PROGRAM MOTORS
VAR
	
END_VAR

Axis_MAIN(sName:='MAIN');
Axis_SUPPLY(sNAme:='SUPPLY');
Axis_JACK1(sNAme:='JACK1');

END_PROGRAM

(* stored: Version 1.1.0.1, ProductVersion 3.1.4024.12
   POU MOTORS: Id {16a50c5a-79ce-4927-aa8a-38fc0bc20c74}, SpecialFunc None *)
